// TIA Portal V18 export
// export: Created 2026-06-08T16:04:38.1869436Z, ExportSetting WithDefaults, DisplayName Totally Integrated Automation Portal, DisplayVersion V18, DisplayName TIA Portal Openness, DisplayVersion V18, DisplayName TIA Portal Version Control Interface, DisplayVersion V18, DisplayName STEP 7 Professional, DisplayVersion V18, DisplayName STEP 7 Safety, DisplayVersion V18, DisplayName WinCC Professional, DisplayVersion V18
FUNCTION "FC_AUTO_MODE" : Void   // FC2, LAD
{ S7_Optimized_Access := 'TRUE' }
VERSION : 0.1
// stored: AutoNumber true, IsIECCheckEnabled false, SetENOAutomatically false, UDAEnableTagReadback false
   VAR_TEMP   // added for the SCL form of the ladder/FBD networks
      _w1 : Bool;
      _w2 : Bool;
      _w3 : Bool;
      _w4 : Bool;
      _w5 : Bool;
      _w6 : Bool;
   END_VAR
BEGIN

REGION Network 1: RESET CÁC BỘ ĐẾM VỀ 0
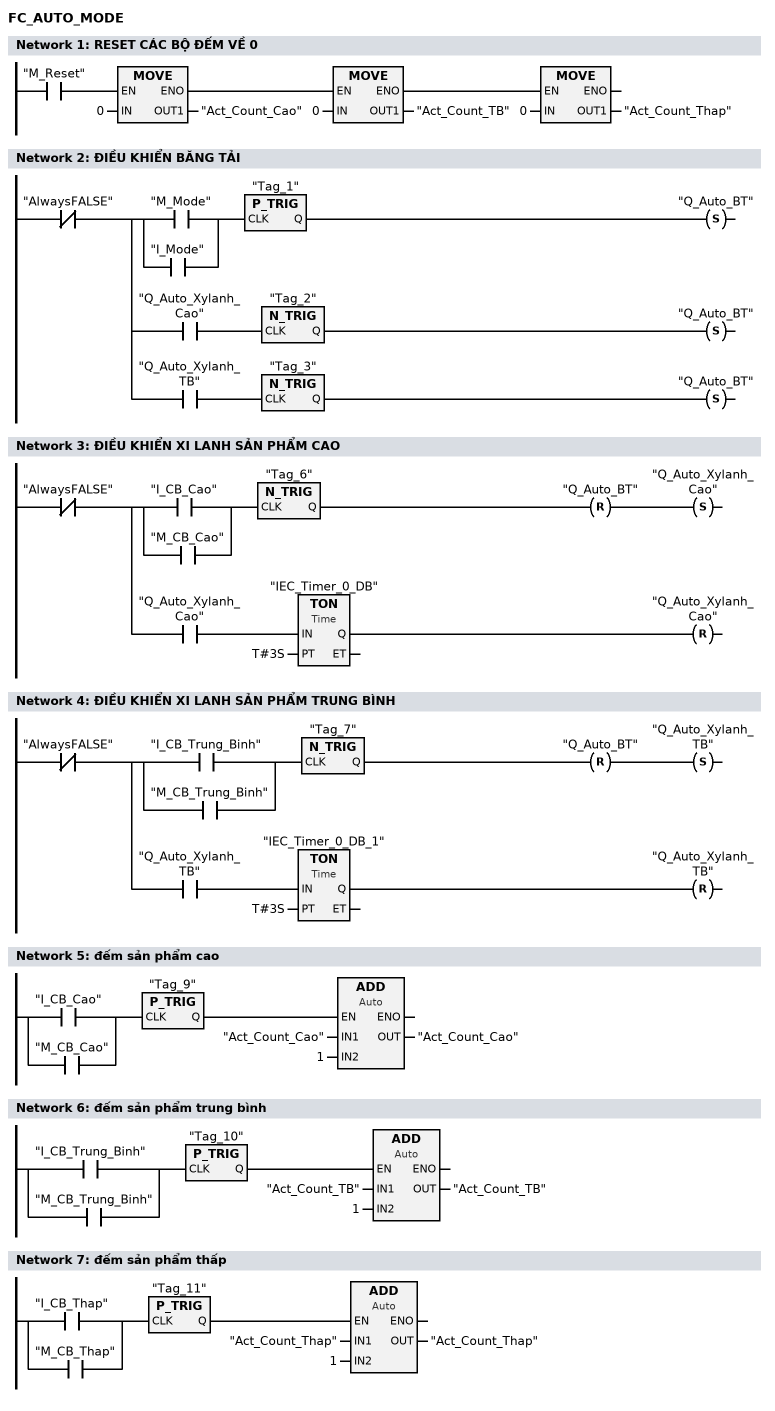
   RUNG wire#powerrail
      Contact( "M_Reset" )
      Move(in := 0, out1 => "Act_Count_Cao")
      Move(in := 0, out1 => "Act_Count_TB")
      Move(in := 0, out1 => "Act_Count_Thap")
   END_RUNG
   // the same network as SCL:
   IF "M_Reset" THEN
       "Act_Count_Cao" := 0;
       "Act_Count_TB" := 0;
       "Act_Count_Thap" := 0;
   END_IF;
END_REGION

REGION Network 2: ĐIỀU KHIỂN BĂNG TẢI
   RUNG wire#powerrail
      I_Contact( "AlwaysFALSE" )
      wire#w1
      Contact( "M_Mode" )
      wire#w2
      P_Trig( "Tag_1" )
      S_Coil( "Q_Auto_BT" )
   END_RUNG
   RUNG wire#w1
      Contact( "I_Mode" )
   END_RUNG wire#w2
   RUNG wire#w1
      Contact( "Q_Auto_Xylanh_Cao" )
      N_Trig( "Tag_2" )
      S_Coil( "Q_Auto_BT" )
   END_RUNG
   RUNG wire#w1
      Contact( "Q_Auto_Xylanh_TB" )
      N_Trig( "Tag_3" )
      S_Coil( "Q_Auto_BT" )
   END_RUNG
   // the same network as SCL:
   #_w1 := NOT "AlwaysFALSE" AND ("M_Mode" OR "I_Mode");
   #_w2 := #_w1 AND NOT "Tag_1";   // rising edge
   "Tag_1" := #_w1;
   IF #_w2 THEN "Q_Auto_BT" := TRUE; END_IF;
   #_w3 := NOT "AlwaysFALSE" AND "Q_Auto_Xylanh_Cao";
   #_w4 := NOT #_w3 AND "Tag_2";   // falling edge
   "Tag_2" := #_w3;
   IF #_w4 THEN "Q_Auto_BT" := TRUE; END_IF;
   #_w5 := NOT "AlwaysFALSE" AND "Q_Auto_Xylanh_TB";
   #_w6 := NOT #_w5 AND "Tag_3";   // falling edge
   "Tag_3" := #_w5;
   IF #_w6 THEN "Q_Auto_BT" := TRUE; END_IF;
END_REGION

REGION Network 3: ĐIỀU KHIỂN XI LANH SẢN PHẨM CAO
   RUNG wire#powerrail
      I_Contact( "AlwaysFALSE" )
      wire#w1
      Contact( "I_CB_Cao" )
      wire#w2
      N_Trig( "Tag_6" )
      R_Coil( "Q_Auto_BT" )
      S_Coil( "Q_Auto_Xylanh_Cao" )
   END_RUNG
   RUNG wire#w1
      Contact( "M_CB_Cao" )
   END_RUNG wire#w2
   RUNG wire#w1
      Contact( "Q_Auto_Xylanh_Cao" )
      { S7_Templates := "time_type := Time" } "IEC_Timer_0_DB".TON(pt := T#3S, et =>)
      R_Coil( "Q_Auto_Xylanh_Cao" )
   END_RUNG
   // the same network as SCL:
   #_w1 := NOT "AlwaysFALSE" AND ("I_CB_Cao" OR "M_CB_Cao");
   #_w2 := NOT #_w1 AND "Tag_6";   // falling edge
   "Tag_6" := #_w1;
   IF #_w2 THEN
       "Q_Auto_BT" := FALSE;
       "Q_Auto_Xylanh_Cao" := TRUE;
   END_IF;
   "IEC_Timer_0_DB".TON(IN := NOT "AlwaysFALSE" AND "Q_Auto_Xylanh_Cao", PT := T#3S);
   IF "IEC_Timer_0_DB".Q THEN "Q_Auto_Xylanh_Cao" := FALSE; END_IF;
END_REGION

REGION Network 4: ĐIỀU KHIỂN XI LANH SẢN PHẨM TRUNG BÌNH
   RUNG wire#powerrail
      I_Contact( "AlwaysFALSE" )
      wire#w1
      Contact( "I_CB_Trung_Binh" )
      wire#w2
      N_Trig( "Tag_7" )
      R_Coil( "Q_Auto_BT" )
      S_Coil( "Q_Auto_Xylanh_TB" )
   END_RUNG
   RUNG wire#w1
      Contact( "M_CB_Trung_Binh" )
   END_RUNG wire#w2
   RUNG wire#w1
      Contact( "Q_Auto_Xylanh_TB" )
      { S7_Templates := "time_type := Time" } "IEC_Timer_0_DB_1".TON(pt := T#3S, et =>)
      R_Coil( "Q_Auto_Xylanh_TB" )
   END_RUNG
   // the same network as SCL:
   #_w1 := NOT "AlwaysFALSE" AND ("I_CB_Trung_Binh" OR "M_CB_Trung_Binh");
   #_w2 := NOT #_w1 AND "Tag_7";   // falling edge
   "Tag_7" := #_w1;
   IF #_w2 THEN
       "Q_Auto_BT" := FALSE;
       "Q_Auto_Xylanh_TB" := TRUE;
   END_IF;
   "IEC_Timer_0_DB_1".TON(IN := NOT "AlwaysFALSE" AND "Q_Auto_Xylanh_TB", PT := T#3S);
   IF "IEC_Timer_0_DB_1".Q THEN "Q_Auto_Xylanh_TB" := FALSE; END_IF;
END_REGION

REGION Network 5: đếm sản phẩm cao
   RUNG wire#powerrail
      Contact( "I_CB_Cao" )
      wire#w1
      P_Trig( "Tag_9" )
      Add(in1 := "Act_Count_Cao", in2 := 1, out => "Act_Count_Cao")
   END_RUNG
   RUNG wire#powerrail
      Contact( "M_CB_Cao" )
   END_RUNG wire#w1
   // the same network as SCL:
   #_w1 := "I_CB_Cao" OR "M_CB_Cao";
   #_w2 := #_w1 AND NOT "Tag_9";   // rising edge
   "Tag_9" := #_w1;
   IF #_w2 THEN "Act_Count_Cao" := "Act_Count_Cao" + 1; END_IF;
END_REGION

REGION Network 6: đếm sản phẩm trung bình
   RUNG wire#powerrail
      Contact( "I_CB_Trung_Binh" )
      wire#w1
      P_Trig( "Tag_10" )
      Add(in1 := "Act_Count_TB", in2 := 1, out => "Act_Count_TB")
   END_RUNG
   RUNG wire#powerrail
      Contact( "M_CB_Trung_Binh" )
   END_RUNG wire#w1
   // the same network as SCL:
   #_w1 := "I_CB_Trung_Binh" OR "M_CB_Trung_Binh";
   #_w2 := #_w1 AND NOT "Tag_10";   // rising edge
   "Tag_10" := #_w1;
   IF #_w2 THEN "Act_Count_TB" := "Act_Count_TB" + 1; END_IF;
END_REGION

REGION Network 7: đếm sản phẩm thấp
   RUNG wire#powerrail
      Contact( "I_CB_Thap" )
      wire#w1
      P_Trig( "Tag_11" )
      Add(in1 := "Act_Count_Thap", in2 := 1, out => "Act_Count_Thap")
   END_RUNG
   RUNG wire#powerrail
      Contact( "M_CB_Thap" )
   END_RUNG wire#w1
   // the same network as SCL:
   #_w1 := "I_CB_Thap" OR "M_CB_Thap";
   #_w2 := #_w1 AND NOT "Tag_11";   // rising edge
   "Tag_11" := #_w1;
   IF #_w2 THEN "Act_Count_Thap" := "Act_Count_Thap" + 1; END_IF;
END_REGION
END_FUNCTION
